FUNCTION_BLOCK Corazon
VAR_INPUT
END_VAR
VAR_OUTPUT
END_VAR
VAR
	VarHumano: Humano;
	pHumano: POINTER TO Humano;
	pHumano16: REFERENCE TO Humano;
END_VAR

END_FUNCTION_BLOCK

(* stored: Version 1.1.0.1, ProductVersion 3.1.4024.12
   POU Corazon: Id {2ac7dfa3-56a7-4936-b4e8-6ace6572c042}, SpecialFunc None *)
